(* IEC 61131-3 sources: RL_MAR/experiments/comparison/llm4plc/results/gpt-4o-mini_20260506_100619/20260506_102702, 2 files *)

(* ---- generated_code_iteration_0.st ---- *)
ructured-text
START_ST
FUNCTION_BLOCK PouchMachine
VAR_INPUT
    start_machine: BOOL;
    stop_machine: BOOL;
END_VAR

VAR_OUTPUT
    machine_ready: BOOL;
    feeder_running: BOOL;
    cutter_running: BOOL;
    heating_running: BOOL;
    cooling_running: BOOL;
END_VAR

VAR
    state: INT := 0; // THE STATE VARIABLE
    prevState: INT := 0; // THE PREVIOUS STATE VARIABLE
    startup_complete: BOOL := FALSE; // INDICATES IF STARTUP IS COMPLETE
    shutdown_complete: BOOL := FALSE; // INDICATES IF SHUTDOWN IS COMPLETE
    heater_status: ARRAY[1..8] OF BOOL; // STATUS OF HEATING STATIONS
    cooler_status: ARRAY[1..8] OF BOOL; // STATUS OF COOLING STATIONS
    feeder_status: BOOL; // STATUS OF FEEDERS
    cutter_status: BOOL; // STATUS OF CUTTERS
    winding_tension: BOOL; // STATUS OF WINDING TENSION
END_VAR

// STATE MACHINE LOGIC
CASE state OF
    0: // INITIALIZE
        machine_ready := FALSE;
        feeder_running := FALSE;
        cutter_running := FALSE;
        heating_running := FALSE;
        cooling_running := FALSE;

        IF start_machine THEN
            state := 1; // Transition to STARTUP SEQUENCE
        END_IF;

    1: // STARTUP SEQUENCE
        FOR i := 1 TO 8 DO
            heater_status[i] := TRUE; // Activate heating stations
            cooler_status[i] := TRUE; // Activate cooling stations
        END_FOR;

        feeder_status := TRUE; // Start feeders
        winding_tension := TRUE; // Establish winding tension

        startup_complete := TRUE; // Set startup_complete to TRUE

        IF startup_complete THEN
            state := 2; // Transition to RUNNING
        END_IF;

    2: // RUNNING
        machine_ready := TRUE;
        feeder_running := TRUE;
        cutter_running := TRUE;
        heating_running := TRUE;
        cooling_running := TRUE;

        IF stop_machine THEN
            state := 3; // Transition to SHUTDOWN SEQUENCE
        END_IF;

    3: // SHUTDOWN SEQUENCE
        cutter_status := FALSE; // Stop cutters
        feeder_status := FALSE; // Stop feeders

        FOR i := 1 TO 8 DO
            heater_status[i] := FALSE; // Deactivate heating stations
            cooler_status[i] := FALSE; // Deactivate cooling stations
        END_FOR;

        shutdown_complete := TRUE; // Set shutdown_complete to TRUE

        IF shutdown_complete THEN
            state := 4; // Transition to NOT READY
        END_IF;

    4: // NOT READY
        machine_ready := FALSE;
        feeder_running := FALSE;
        cutter_running := FALSE;
        heating_running := FALSE;
        cooling_running := FALSE;

        // Optionally, reset state to INITIALIZE if needed
        // state := 0;
END_CASE;

END_FUNCTION_BLOCK
END_ST

(* ---- generated_code_iteration_1.st ---- *)
START_REASON
The errors in the original Structured Text (ST) code occurred because the variable 'i' was not defined before it was used in the FOR loop. In ST, all loop control variables must be declared in the VAR section before they can be utilized. This oversight led to the compiler error indicating that the identifier 'i' was not defined. To resolve this, I will declare 'i' as an integer variable in the VAR section before it is used in the FOR loop.
END_REASON

START_ST
FUNCTION_BLOCK PouchMachine
VAR_INPUT
    start_machine: BOOL;
    stop_machine: BOOL;
END_VAR

VAR_OUTPUT
    machine_ready: BOOL;
    feeder_running: BOOL;
    cutter_running: BOOL;
    heating_running: BOOL;
    cooling_running: BOOL;
END_VAR

VAR
    state: INT := 0; // THE STATE VARIABLE
    prevState: INT := 0; // THE PREVIOUS STATE VARIABLE
    startup_complete: BOOL := FALSE; // INDICATES IF STARTUP IS COMPLETE
    shutdown_complete: BOOL := FALSE; // INDICATES IF SHUTDOWN IS COMPLETE
    heater_status: ARRAY[1..8] OF BOOL; // STATUS OF HEATING STATIONS
    cooler_status: ARRAY[1..8] OF BOOL; // STATUS OF COOLING STATIONS
    feeder_status: BOOL; // STATUS OF FEEDERS
    cutter_status: BOOL; // STATUS OF CUTTERS
    winding_tension: BOOL; // STATUS OF WINDING TENSION
    i: INT; // LOOP CONTROL VARIABLE
END_VAR

// STATE MACHINE LOGIC
CASE state OF
    0: // INITIALIZE
        machine_ready := FALSE;
        feeder_running := FALSE;
        cutter_running := FALSE;
        heating_running := FALSE;
        cooling_running := FALSE;

        IF start_machine THEN
            state := 1; // Transition to STARTUP SEQUENCE
        END_IF;

    1: // STARTUP SEQUENCE
        FOR i := 1 TO 8 DO
            heater_status[i] := TRUE; // Activate heating stations
            cooler_status[i] := TRUE; // Activate cooling stations
        END_FOR;

        feeder_status := TRUE; // Start feeders
        winding_tension := TRUE; // Establish winding tension

        startup_complete := TRUE; // Set startup_complete to TRUE

        IF startup_complete THEN
            state := 2; // Transition to RUNNING
        END_IF;

    2: // RUNNING
        machine_ready := TRUE;
        feeder_running := TRUE;
        cutter_running := TRUE;
        heating_running := TRUE;
        cooling_running := TRUE;

        IF stop_machine THEN
            state := 3; // Transition to SHUTDOWN SEQUENCE
        END_IF;

    3: // SHUTDOWN SEQUENCE
        cutter_status := FALSE; // Stop cutters
        feeder_status := FALSE; // Stop feeders

        FOR i := 1 TO 8 DO
            heater_status[i] := FALSE; // Deactivate heating stations
            cooler_status[i] := FALSE; // Deactivate cooling stations
        END_FOR;

        shutdown_complete := TRUE; // Set shutdown_complete to TRUE

        IF shutdown_complete THEN
            state := 4; // Transition to NOT READY
        END_IF;

    4: // NOT READY
        machine_ready := FALSE;
        feeder_running := FALSE;
        cutter_running := FALSE;
        heating_running := FALSE;
        cooling_running := FALSE;

        // Optionally, reset state to INITIALIZE if needed
        // state := 0;
END_CASE;

END_FUNCTION_BLOCK
END_ST
